// TwinCAT 3 PLC project PLC_BMS
// ProgramVersion: 3.1.4026.12
// libraries:
//   Tc2_ModbusSrv, * (Beckhoff Automation GmbH)
//   Tc2_Standard, * (Beckhoff Automation GmbH)
//   Tc2_System, * (Beckhoff Automation GmbH)
//   Tc2_Utilities, * (Beckhoff Automation GmbH)
//   Tc3_IotBase, * (Beckhoff Automation GmbH)
//   Tc3_Module, * (Beckhoff Automation GmbH)
// project tree:
//   DUTs/ BessOpmodeControl.TcDUT, BessStateControl.TcDUT, DATAEXCH.TcDUT, Ethercat_AlarmsWarningToCLC.TcDUT, EtherCAT_Monitor_BatVariables.TcDUT, MBCommandsFrmCLC.TcDUT, EtherCATCommandsFrmCLC.TcDUT, ETherCAT_StatMonitor_VAR.TcDUT, ModbusRead.TcDUT, ModbusWrite.TcDUT, StateMachineCommand.TcDUT, MB_StatMonitoring_VAR.TcDUT, EtherCAT_Parameters_FrmCLC.TcDUT
//   / GlobalTextList.TcGTLO, ModbusTask.TcTTO, StateMachineTask.TcTTO
//   GVLs/ GVL_Global.TcGVL
//   POUs/ DataLogic.TcPOU, MAIN.TcPOU, ModbusControl.TcPOU, StateMachine.TcPOU
// real-time tasks:
//   TASK ModbusTask: cycle T#20ms, priority 8, ADS port 352
//   TASK StateMachineTask: cycle T#5ms, priority 6, ADS port 350
// I/O:
//   DEVICE Device 1 (EtherCAT Slave), AmsNetId 10.200.8.4.2.255
// variable links:
//   PLC-BMS/PLC-BMS Instance <-> Device 1 (EtherCAT Slave)
//     ModbusTask Inputs/GVL_Global.EthercatParametersIN <-> Inputs/ParametersIN
//     ModbusTask Inputs/GVL_Global.udev <-> InfoData/State
//     ModbusTask Outputs/GVL_Global.EthercatMoniotrBAT_OUT <-> Outputs/EthercatMonitorBatVarOUT
//     ModbusTask Outputs/GVL_Global.EthercatSTATMonitoringOut <-> Outputs/StatMonitorVarOut
//     ModbusTask Outputs/GVL_Global.Ethercat_alarms_warningsOUT <-> Outputs/AlarmsWarningOUT
//     ModbusTask Outputs/GVL_Global.test <-> Outputs/Var 11
//     StateMachineTask Inputs/GVL_Global.EthCommandsfrmCLC_IN <-> Inputs/CommanndsfromCLC
//     StateMachineTask Inputs/GVL_Global.data2rcv <-> Inputs/data2rcv

CONFIGURATION PLC_BMS
    RESOURCE PLC ON TwinCAT3
        TASK ModbusTask(INTERVAL := T#20ms, PRIORITY := 8);
        TASK StateMachineTask(INTERVAL := T#5ms, PRIORITY := 6);
        PROGRAM ModbusControl WITH ModbusTask : ModbusControl;
        PROGRAM StateMachine WITH StateMachineTask : StateMachine;
        PROGRAM MAIN WITH StateMachineTask : MAIN;
        PROGRAM DataLogic WITH StateMachineTask : DataLogic;
    END_RESOURCE
END_CONFIGURATION

// ---- DUTs/BessOpmodeControl.TcDUT
{attribute 'qualified_only'}

TYPE BessOpmodeControl :
(
	OPERATIONAL := 1, // P/Q Connected to grid and injecting current
	DISCONNECTED := 2,   // OFF-grid Disoconneted from grid
	CONNECTED := 3 // On-grid Connected to grid but no injection
	
)UINT;
END_TYPE

// ---- DUTs/BessStateControl.TcDUT
{attribute 'qualified_only'}
{attribute 'strict'}
TYPE BessStateControl :
(
	STOP := 2,
	RUN := 6
)UINT;
END_TYPE

// ---- DUTs/DATAEXCH.TcDUT
TYPE DATAEXCH :
STRUCT
cmd : ARRAY [0..10] OF INT ;
param 	: ARRAY [0..10] OF REAL ;
variables: ARRAY [0..100] OF REAL ;
statVAR: ARRAY [0..20] OF REAL ;

END_STRUCT
END_TYPE

// ---- DUTs/Ethercat_AlarmsWarningToCLC.TcDUT
TYPE Ethercat_AlarmsWarningToCLC :
STRUCT
	Communication_Alarms : BOOL; 
	Battery_Alarms : BOOL;
	Warnings: BOOL;
	Faults: BOOL;
	reservebit1 : BOOL;
	reservebit2 : BOOL;
	reservebit3 : BOOL;
	reservebit4 : BOOL;

END_STRUCT
END_TYPE

// ---- DUTs/EtherCAT_Monitor_BatVariables.TcDUT
TYPE EtherCAT_Monitor_BatVariables :
STRUCT

	
VaRMS 	:REAL;
VbRMS	:REAL;
VcRMS	:REAL;
IaRMS	:REAL;
IbRMS	:REAL;
IcRMS	:REAL;
Total_ActivePower	:REAL;
Total_ReactivePower	:REAL;
Grid_Frequency	:REAL;
PowerFactor	:REAL;
Vdc	:REAL;
Idc	:REAL;
SoC	:REAL;
SoH	:REAL; 
reserve1: REAL;
reserve2: REAL;

END_STRUCT
END_TYPE

// ---- DUTs/MBCommandsFrmCLC.TcDUT
TYPE MBCommandsFrmCLC :
STRUCT
	//Commands from CLC  read at output register CLC master
	//state control enum type. 
	commands : StateMachineCommand;
	
	//P Q references. 
	ActivePowerReference : DINT;
	ReactivePowerReferecne: DINT;
	Heartbeat : DINT;
	ClrAlarm : DINT;
	ClrFault : DINT;
	
	
END_STRUCT
END_TYPE

// ---- DUTs/EtherCATCommandsFrmCLC.TcDUT
TYPE EtherCATCommandsFrmCLC :
STRUCT
	//Commands from CLC  ETHERCAT IN
	//state control enum type. 
	StatControlCMD : BessStateControl;
	OpModeControlCMD : BessOpmodeControl;
	//P Q references. 
	ActivePowerReference : DINT;
	ReactivePowerReference: DINT;
	Heartbeat : DINT;
	ClrAlarm : DINT;
	ClrFault : DINT;
	reserve1 : DINT;
	reserver2 : DINT;
	
	
	
	
END_STRUCT
END_TYPE

// ---- DUTs/ETherCAT_StatMonitor_VAR.TcDUT
TYPE ETherCAT_StatMonitor_VAR :
STRUCT
	//variables to be monitored // EthererCAT out  (IN for CLC)
	
	StatControlCMD : BessStateControl;
	OpModeControlCMD : BessOpmodeControl;
	//P Q references. 
	ActivePowerReference : DINT;
	ReactivePowerReference: DINT;
	Heartbeat : DINT;
	ClrAlarm : DINT;
	ClrFault : DINT;
	reserve1 : DINT;
	reserver2 : DINT;
	

		
END_STRUCT
END_TYPE

// ---- DUTs/ModbusRead.TcDUT
TYPE ModbusRead : // EnerArk 
STRUCT

Workingstatus	:USINT; //0x0001

Workingmode	:USINT;

Controlmode	:USINT;

Allowable_discharge_active_powerlimit	:USINT;

Allowable_charging_active_powerlimit	:USINT;

System_active_power	:USINT;

Load_active_power	:INT;

Grid_active_power	:INT;

MPPT_total_power	:USINT;
grid_input_active_powerHigh	:USINT;

grid_input_active_powerLow	:USINT;

grid_output_active_powerHigh	:USINT;

grid_output_active_powerLow	:USINT;

Load_output_active_powerHigh	:USINT;

Load_output_active_powerLow :USINT;

UC1_working_status	:USINT;

UC2_working_status	:USINT;

UC3_working_status	:USINT;

UC4_working_status	:USINT;

UC5_working_status	:USINT;

UC6_working_status	:USINT;

UC7_working_status	:USINT;

UC8_working_status	:USINT;

UC9_working_status	:USINT;

UC10_working_status	:USINT;

Reserved	:USINT;

System_alarm0	:USINT;

System_alarm1	:USINT;

System_failure0	:USINT;

System_failure1	:USINT; //0x001E



END_STRUCT
END_TYPE

// ---- DUTs/ModbusWrite.TcDUT

TYPE ModbusWrite :
STRUCT
		
System_mode_control	: BessOpmodeControl; ///USINT; //0x003c

System_state_control	: BessStateControl; //USINT;

Control_mode	:USINT;

Active_power_control	: INT := 0;  //init

Reactive_power_control	: INT := 0; //init

SOC_H	:USINT;
SOC_L	:USINT;

Backu_charging_power	:USINT;

Initial_operating_mode	:USINT;

Initial_control_mode	:USINT;

Slave_address	:USINT;

Rated_power	:USINT;

Clear_fault	:USINT; // 0x0048

END_STRUCT
END_TYPE

// ---- DUTs/StateMachineCommand.TcDUT
{attribute 'qualified_only'}
{attribute 'strict'}
{attribute 'to_string'}
TYPE StateMachineCommand  :
(
	OFF := 0,
	DISCONNECTED:= 1,
	CONNECTED := 2,
	OPERATIONAL := 3,
	FAULT := 4
) INT;
END_TYPE

// ---- DUTs/MB_StatMonitoring_VAR.TcDUT
TYPE MB_StatMonitoring_VAR :
STRUCT
	//variables to be monitored // write to CLC master output register
	
	// Status related 
	CurrentOpmod : StateMachineCommand;
	
	// HEATBIT , 	
	Heartbeat : DINT; // An inc. counter
	
	Alarms1 : DINT;  
	Alarms2: DINT;  
	
	Alarms3 : DINT;
	Alarms4  : DINT;  	

	Warning1 :DINT;
	Warning2: DINT;
	
	

		
END_STRUCT
END_TYPE

// ---- DUTs/EtherCAT_Parameters_FrmCLC.TcDUT
TYPE EtherCAT_Parameters_FrmCLC :
STRUCT
	//set from CLC(commuinity level controller  )
	MIN_SoC : REAL;
	MAX_SoC :  REAL;
	P_LIMIT :  REAL;
	Q_LIMIT:  REAL;
	ChargeRate_LIMIT:  REAL;
	DischargeRate_LIMIT:  REAL;
	Initial_Energy:  REAL;
	Terminal_Energy:  REAL;

END_STRUCT
END_TYPE

// ---- GVLs/GVL_Global.TcGVL
{attribute 'qualified_only'}
VAR_GLOBAL
	bON : BOOL;
	bOFF: BOOL;
	bDisconnected: BOOL;
	bConnected: BOOL;
	bOPERATIONAL: BOOL;
	bFault_present: BOOL;
	bAlarm_present: BOOL;
	bCommunicationOK: BOOL :=TRUE;
	bClearFault: BOOL;
	bClearAlarm: BOOL;
	
	ModRead : ModbusRead;
	ModWrite : ModbusWrite;
	bPower_enable : BOOL;
	
	//Data Excahnge 
	//data2send AT %Q* : DATAEXCH;
	data2rcv AT %I* : DATAEXCH;
	
	
	
	EthercatParametersIN AT %I* : EtherCAT_Parameters_FrmCLC;
	EthCommandsfrmCLC_IN AT %I* : EtherCATCommandsFrmCLC; // command from clc on Ethercat
	EthercatSTATMonitoringOut AT %Q* :ETherCAT_StatMonitor_VAR; //status var for clc on Ethercat
	EthercatMoniotrBAT_OUT AT %Q* : EtherCAT_Monitor_BatVariables;
	Ethercat_alarms_warningsOUT AT %Q* : Ethercat_AlarmsWarningToCLC;
	
	monitoringVAR : MB_StatMonitoring_VAR;  //send to CLC master modbus test
	commandsfromCLC : MBCommandsFrmCLC; //modbus link to clc master
	
	udev AT %I*: UINT;
	test AT %Q* : DINT;
	data : ARRAY [0..4] OF WORD;
	enstate : INT ;
	CommunicationFailureEtherCAT : BOOL;
END_VAR

// ---- POUs/ModbusControl.TcPOU
PROGRAM ModbusControl
VAR
	bWrite : BOOL;
	bRead: BOOL;
	fbMBwritereg : FB_MBWriteRegs;  
	fbMBreadreg : FB_MBReadRegs;
	adata : ARRAY [0..3] OF WORD;
	adatar : ARRAY [0..3] OF WORD;
	nQ : WORD :=4;
	estateread : StateMachineCommand;
	
	
END_VAR

GVL_Global.monitoringVAR.CurrentOpmod :=GVL_Global.commandsfromCLC.commands;
//GVL_Global.ModWrite.System_state_control  := GVL_Global.EthCommandsfrmCLC_IN.StatControlCMD;
GVL_Global.ModWrite.System_mode_control  := GVL_Global.EthCommandsfrmCLC_IN.OpModeControlCMD;
IF GVL_Global.bPower_enable = TRUE THEN
GVL_Global.ModWrite.Active_power_control := DINT_TO_INT(GVL_Global.EthCommandsfrmCLC_IN.ActivePowerReference)*10;
GVL_Global.ModWrite.Reactive_power_control := DINT_TO_INT(GVL_Global.EthCommandsfrmCLC_IN.ReactivePowerReference)*10;
ELSE
	GVL_Global.ModWrite.Active_power_control := 0;
GVL_Global.ModWrite.Reactive_power_control :=0;
END_IF
GVL_Global.ModWrite.Clear_fault := DINT_TO_USINT(GVL_Global.EthCommandsfrmCLC_IN.ClrFault);

IF NOT fbMBwritereg.bBusy THEN
	bWrite := TRUE;
fbMBwritereg(
	sIPAddr:= '10.200.8.219', //write at output reg of master i.e Eneraerk , CLC -- ws2lc
	nTCPPort:= 502, 
	nUnitID:= 255, 
	nQuantity:=SIZEOF(GVL_Global.ModWrite)/2, 
	nMBAddr:= 16#8020, 
	cbLength:= SIZEOF(GVL_Global.ModWrite), 
	pSrcAddr:= ADR(GVL_Global.ModWrite), 
	bExecute:= bWrite, 
	tTimeout:= T#5S, 
	bBusy=> , 
	bError=> , 
	nErrId=> );
	ELSE
		bWrite:= FALSE;
		fbMBwritereg(bExecute :=bWrite);
		
	END_IF
	
	IF NOT fbMBreadreg.bBusy THEN
		bRead := TRUE;
	fbMBreadreg(
	sIPAddr:= '10.200.8.219', 
	nTCPPort:= 502, 
	nUnitID:= 255, 
	nQuantity:= SIZEOF(GVL_Global.ModRead)/2, 
	nMBAddr:= 16#8000, 
	cbLength:= SIZEOF(GVL_Global.ModRead), 
	pDestAddr:= ADR(GVL_Global.ModRead), 
	bExecute:= bRead, 
	tTimeout:= T#5S, 
	bBusy=> , 
	bError=> , 
	nErrId=> , 
	cbRead=> );
	ELSE
		bRead := FALSE;
		fbMBreadreg(bExecute := bRead);
		
	END_IF
	//GVL_Higherlevel.enstate := WORD_TO_INT(adatar[0]);

END_PROGRAM

// ---- POUs/StateMachine.TcPOU
PROGRAM StateMachine
VAR
	eFLCState: StateMachineCommand;
	params_fromHL : EtherCAT_Parameters_FrmCLC; //param from high /2nd level
	sCurrentState: STRING;
	sAlarm: STRING;
	
	tRamping :  TOF := (PT:=T#2S);
	sRamping: STRING;
	EtherCATHeartBeat : DINT;
	CounterCommFailure : INT;
END_VAR

// Protection for EtherCAT
//EtherCATHeartBeat := EtherCATHeartBeat+1;
	IF GVL_Global.EthCommandsfrmCLC_IN.Heartbeat = EtherCATHeartBeat THEN
		CounterCommFailure := CounterCommFailure + 1;
			IF CounterCommFailure > 500 THEN
				 GVL_Global.EthCommandsfrmCLC_IN.StatControlCMD:= 2;
				GVL_Global.CommunicationFailureEtherCAT := TRUE;
				//Communications.EtherCAT_Variables.WarningLog.Bits.EtherCAT_Failure := TRUE;
				CounterCommFailure := 0;
			END_IF
	ELSE
		GVL_Global.CommunicationFailureEtherCAT:= FALSE;
		//Communications.EtherCAT_Variables.WarningLog.Bits.EtherCAT_Failure := FALSE;
		CounterCommFailure := 0;
	END_IF
	EtherCATHeartBeat := GVL_Global.EthCommandsfrmCLC_IN.Heartbeat ;

//FLC State machine goverened by state of Enerark BESS EMS modbus module	
IF GVL_Global.ModRead.Workingstatus = 1 OR GVL_Global.ModWrite.System_state_control =2 THEN   // 1 = stop, 2 =  run, 3 = fault,   MB register work_status address 0x001
eFLCState := StateMachineCommand.OFF;
ELSIF GVL_Global.ModRead.Workingstatus = 2 OR GVL_Global.ModWrite.System_state_control = 6 THEN
	IF GVL_Global.ModRead.Workingmode = 1 OR GVL_Global.ModWrite.System_mode_control = 1 THEN     // 1 = P/Q , 2 = off-grid, 3 = on-grid? 4 = peak to valley mode 5= backup mode
		eFLCState := StateMachineCommand.OPERATIONAL;
		ELSIF GVL_Global.ModRead.Workingmode = 2 OR GVL_Global.ModWrite.System_mode_control =2 THEN
			eFLCState := StateMachineCommand.DISCONNECTED;
			ELSIF GVL_Global.ModRead.Workingmode = 3 OR GVL_Global.ModWrite.System_mode_control = 3 THEN
				eFLCState := StateMachineCommand.CONNECTED;
				END_IF
	ELSIF GVL_Global.ModRead.Workingstatus = 3 THEN
		eFLCState := StateMachineCommand.FAULT;
		END_IF	

CASE eFLCState OF
	
	//Default satate after switching on controller.
	StateMachineCommand.OFF:
		GVL_Global.bPower_enable := FALSE;
		//GVL_Global.ModWrite.Active_power_control := 0;
		//GVL_Global.ModWrite.Reactive_power_control := 0;
	
		(*//commuincation check , INIT
		IF GVL_Global.bCommunicationOK THEN
			IF GVL_Global.bON AND NOT GVL_Global.bOFF THEN
				eFLCState := StateMachineCommand.DISCONNECTED;
			END_IF
					
		END_IF*)
	
	// BESS is ready but not connected to GRID
	StateMachineCommand.DISCONNECTED:
		GVL_Global.bPower_enable := FALSE;
		//GVL_Global.ModWrite.Active_power_control := 0;
		//GVL_Global.ModWrite.Reactive_power_control := 0;
	
		//check faults/alarms
		(*IF GVL_Global.bFault_present THEN
			eFLCState := StateMachineCommand.FAULT;
	
		ELSE
			IF GVL_Global.bConnected THEN
			eFLCState := StateMachineCommand.CONNECTED;
			END_IF
		END_IF*)
	//BESS is connected to GRID but no Injection
	StateMachineCommand.CONNECTED:
		GVL_Global.bPower_enable := FALSE;
		//GVL_Global.ModWrite.Active_power_control := 0;
		//GVL_Global.ModWrite.Reactive_power_control := 0;
	
		(*IF GVL_Global.bFault_present THEN
			eFLCState := StateMachineCommand.FAULT;
	
		ELSE
			IF GVL_Global.bOPERATIONAL THEN
				eFLCState := StateMachineCommand.OPERATIONAL;
			END_IF
			IF NOT GVL_Global.bConnected THEN
				eFLCState := StateMachineCommand.DISCONNECTED;
			END_IF
		END_IF *)
		
	// BESS IN OPERATIONAL MODE , recieve I/0
	StateMachineCommand.OPERATIONAL:
	 //Control varaibles , references  here , 
	 GVL_Global.bPower_enable := TRUE;
		//GVL_Global.ModWrite.Active_power_control :=  DINT_TO_INT(GVL_Global.EthCommandsfrmCLC_IN.ActivePowerReference)*10; //-600 to 600 kW
		
		//GVL_Global.ModWrite.Reactive_power_control := DINT_TO_INT(GVL_Global.EthCommandsfrmCLC_IN.ReactivePowerReference)*10;
		
		(*IF GVL_Global.bFault_present THEN
			eFLCState := StateMachineCommand.FAULT;
	
		END_IF
		IF NOT GVL_Global.bOPERATIONAL THEN
				eFLCState := StateMachineCommand.CONNECTED;
			END_IF*)	
	
//FAULT STATE // 
	StateMachineCommand.FAULT:
	// RAMDOWN /GRID DSICONECTION //// 
		GVL_Global.ModWrite.Active_power_control := 0;
		GVL_Global.ModWrite.Reactive_power_control := 0;
	
	//Clear faults;
		IF GVL_Global.ModRead.Workingstatus = 2   THEN // OR GVL_Global.ModRead.Workingstatus = 1
			// power ramping down 
			//Transit to disconneted or off
			eFLCState := StateMachineCommand.DISCONNECTED;
			GVL_Global.bFault_present := FALSE;
			GVL_Global.bConnected :=FALSE;
			GVL_Global.bOPERATIONAL :=FALSE;
			//IF GVL_Higherlevel.bClearFault THEN
			//GVL_Higherlevel.bFault_present := FALSE;
		
			//END_IF
		
		END_IF		

END_CASE
	
	
	sCurrentState := TO_STRING(eFLCState); // get state name 
	


(*IF GVL_Global.bAlarm_present THEN
		
	// RAMDOWN IF ALARM STAYS  
		sAlarm := 'An alarm is present';
		ELSIF GVL_Global.bClearAlarm THEN
			sAlarm := '';	
	END_IF
	IF GVL_Global.bOFF THEN
		tRamping(IN:=GVL_Global.bOFF) ;
		sRamping := 'Ramping down process ';
		IF tRamping.Q THEN
			sRamping := 'Ramped Down';
			eFLCState:= StateMachineCommand.OFF; 
			sRamping := '';
		END_IF
		eFLCState:= StateMachineCommand.OFF; 
		
	END_IF*)

END_PROGRAM

// ---- POUs/MAIN.TcPOU
PROGRAM MAIN
VAR
	fbMqttClient :  FB_IotMqttClient;
	bSetParameter: BOOL := TRUE;
	bConnect: BOOL := FALSE;
	fbMessageQueue : FB_IotMqttMessageQueue;
	fbMessage      : FB_IotMqttMessage;
	
	sTopicPub   : STRING(255) := 'MyTopic';
    sPayloadPub : STRING(255);
    i : UDINT;
    fbTimer : TON := (PT:=T#1S);
	
	bSubscribed    : BOOL;
    sTopicSub      : STRING(255) := 'MyTopic';
    
	sTopicRcv      : STRING(255);
    sPayloadRcv    : STRING(255);	
END_VAR

 // set parameters once when connecting to the mqtt broker
IF bSetParameter THEN
    bSetParameter               := FALSE;
    fbMqttClient.sHostName      := 'broker.hivemq.com';
    fbMqttClient.nHostPort      := 1883;
    fbMqttClient.sTopicPrefix   := ''; 
    fbMqttClient.sUserName      := 'User';
    fbMqttClient.sUserPassword  := 'TopSecret'; 
    fbMqttClient.ipMessageQueue := fbMessageQueue;
END_IF

// MQTT client must be triggered cyclically
fbMqttClient.Execute(bConnect);

IF fbMqttClient.bConnected THEN
    IF NOT bSubscribed THEN
        bSubscribed := fbMqttClient.Subscribe(sTopic:=sTopicSub, eQoS:=TcIotMqttQos.AtMostOnceDelivery);
    END_IF
    fbTimer(IN:=TRUE);
    IF fbTimer.Q THEN // publish new payload every second
        fbTimer(IN:=FALSE);
        i := i + 1;
        sPayloadPub := CONCAT('MyMessage', TO_STRING(i));
        fbMqttClient.Publish(    sTopic:= sTopicPub, 
                               pPayload:= ADR(sPayloadPub), nPayloadSize:= LEN2(ADR(sPayloadPub))+1,  
                                eQoS:= TcIotMqttQos.AtMostOnceDelivery, bRetain:= FALSE, bQueue:= FALSE );
    END_IF
	
	IF fbMessageQueue.nQueuedMessages > 0 THEN
    IF fbMessageQueue.Dequeue(fbMessage:=fbMessage) THEN
        fbMessage.GetTopic(pTopic:=ADR(sTopicRcv), nTopicSize:=SIZEOF(sTopicRcv) );
        fbMessage.GetPayload(pPayload:=ADR(sPayloadRcv), nPayloadSize:=SIZEOF(sPayloadRcv), bSetNullTermination:=FALSE);
    END_IF
END_IF
END_IF

END_PROGRAM

// ---- POUs/DataLogic.TcPOU
PROGRAM DataLogic
VAR	

END_VAR

CASE GVL_Global.data2rcv.cmd[0] OF 
	0: 
		GVL_Global.ModWrite.System_state_control:=2;	// Stop command
	1:
		GVL_Global.ModWrite.System_state_control := 6; // RUN command 
		//battry on, 
		
END_CASE

CASE GVL_Global.data2rcv.cmd[1] OF
	0: 
		GVL_Global.ModWrite.System_mode_control := 2; // Disconnected 
	1:
		GVL_Global.ModWrite.System_mode_control := 3; //Connected	
	2:
		GVL_Global.ModWrite.System_mode_control := 1; // Operational	
		
END_CASE

END_PROGRAM

// ---- GlobalTextList.TcGTLO
TEXTLIST GlobalTextList
  339 = '%s'
  673 = 'bON'
  118 = 'Clear fault'
  545 = 'Connect'
  57 = 'Connect GRID'
  685 = 'Connected'
  539 = 'CURRENT STATE'
  170 = 'Enum'
  988 = 'OFF'
  879 = 'OP CONTROL'
  562 = 'Operational'
  304 = 'SATE Enum'
  238 = 'STATE ENUM'
  416 = 'TE'
  232 = 'Test Fault satate'
  444 = 'Test Fault state'
  264 = 'TSATE Enum'
END_TEXTLIST
